FUNCTION_BLOCK XtsMover_TestSuite
VAR
	_TestMoverInterface : I_TcIoXtsXpuMover;
	ThisTestSuite : TestSuite<TestSuiteParameter.MaxTestCount>('C:\ProgramData\Beckhoff\TwinCAT\3.1\Boot\XtsMover_Tests.xml') := (TestSuiteName := 'XtsMover Test Suite');
END_VAR

MoverAcceptsEnableCommand_Test();
MoverAcceptsDisableCommand_Test();
MoverAcceptsGoodGap_Test();
MoverAcceptsModuloBackwardMove_Test();
MoverAcceptsModuloForwardMove_Test();
MoverAcceptsModuloForwardOnlyCommand_Test();
MoverAcceptsNonModuloMoveCommand_Test();
MoverRejectsDisableCommand_Test();
MoverRejectsEnableCommand_Test();
MoverRejectsGapLow_Test();
MoverRejectsHighVeloCommand_Test();
MoverRejectsNegVeloCommand_Test();
MoverRejectsResetWithNoError_Test();
MoverRejectsActivateZeroTrack_Test();
MoverRejectsUnusedHighIndexTrack_Test();
MoverRejectsActivateTrackWhileMoving_Test();
MoverRejectsZeroRefSysWhenMoving_Test();
MoverAcceptsZeroRefSysSet_Test();
MoverRejectsCycleCallWithNoAxisRef_Test();
MoverReportsMovingCorrectly_Test();
MoverReportsMoverOutsidePosWindow_Test();
MoverReportsPositionInWindow_Test();
MoverAcceptsTrackRegistration_Test();
MoverRejectsNullTrackRegister_Test();
MoverRejectsDoubleTrackRegister_Test();
MoverRejectsPosCheckwithNoTrack_Test();
MoverRejectsArriveCommandIfNotLeft_Test();
MoverRejectsArriveCommandIfNoInterface_Test();
MoverRejectsLeaveCommandWithNoInterface_Test();
MoverRejectsLeaveCommandIfMoving_Test();
MoverAcceptsMoverLeaveCommand_Test();
MoverAcceptsArriveCommand_Test();
MoverRejectsAbsMoveToSamePosition();
MoverRejectsModuloMoveToSamePosition();

METHOD MoverAcceptsArriveCommand_Test
VAR_INST
	Expected : BOOL := TRUE;
	Actual	 : BOOL;
END_VAR
VAR
	testMover : stubMover;
END_VAR
IF ThisTestSuite.Test(__POUNAME()).ExecuteTest() THEN
	testMover.MoverXtsIoEnvInterface := _TestMoverInterface;
	Actual := SUCCEEDED(testMover.TriggerMoverArrive());
	ThisTestSuite.Test(__POUNAME()).AssertEqual(Expected, Actual);
END_IF
END_METHOD

METHOD MoverAcceptsDisableCommand_Test
VAR_INST
	Expected : BOOL := TRUE;
	Actual	 : BOOL;
END_VAR
VAR
	testMover : stubMover;
END_VAR
IF ThisTestSuite.Test(__POUNAME()).ExecuteTest() THEN
	testMover.setEnabled();
	Actual := SUCCEEDED( testMover.DisableMover());
	ThisTestSuite.Test(__POUNAME()).AssertEqual(Expected, Actual);
END_IF
END_METHOD

METHOD MoverAcceptsEnableCommand_Test : BOOL
VAR_INST
	Expected : BOOL := TRUE;
	Actual	 : BOOL;
END_VAR
VAR
	testMover : stubMover;
END_VAR
IF ThisTestSuite.Test(__POUNAME()).ExecuteTest() THEN
	testMover.setDisabled();
	Actual := SUCCEEDED( testMover.EnableMover());
	ThisTestSuite.Test(__POUNAME()).AssertEqual(Expected, Actual);
END_IF
END_METHOD

METHOD MoverAcceptsGoodGap_Test : BOOL
VAR_INST
	Expected : mc_lreal := 120.0;
	Actual	 : mc_lreal;
END_VAR
VAR
	testMover : XtsMover;
END_VAR
IF ThisTestSuite.Test(__POUNAME()).ExecuteTest() THEN
	testMover.Gap := 120.0;
	Actual := testMover.Gap;
	ThisTestSuite.Test(__POUNAME()).AssertEqual(Expected, Actual);
END_IF
END_METHOD

METHOD MoverAcceptsModuloBackwardMove_Test
VAR_INST
	Expected : BOOL := TRUE;
	Actual	 : BOOL;
END_VAR
VAR
	testMover : stubMover;
END_VAR
IF ThisTestSuite.Test(__POUNAME()).ExecuteTest() THEN
	testMover.PositiveDirectionOnly := FALSE;
	Actual := testMover.MoveTo(RequiredPosition := - 100.0,
											MoveVelocity := 10.0,
											NonModuloMove := FALSE) = 4;
	ThisTestSuite.Test(__POUNAME()).AssertEqual(Expected, Actual);
END_IF
END_METHOD

METHOD MoverAcceptsModuloForwardMove_Test
VAR_INST
	Expected : BOOL := TRUE;
	Actual	 : BOOL;
END_VAR
VAR
	testMover : stubMover;
END_VAR
IF ThisTestSuite.Test(__POUNAME()).ExecuteTest() THEN
	testMover.PositiveDirectionOnly := FALSE;
	Actual := testMover.MoveTo(RequiredPosition := 100.0,
											MoveVelocity := 10.0,
											NonModuloMove := FALSE) = 3;
	ThisTestSuite.Test(__POUNAME()).AssertEqual(Expected, Actual);
END_IF
END_METHOD

METHOD MoverAcceptsModuloForwardOnlyCommand_Test
VAR_INST
	Expected : BOOL := TRUE;
	Actual	 : BOOL;
END_VAR
VAR
	testMover : stubMover;
END_VAR
IF ThisTestSuite.Test(__POUNAME()).ExecuteTest() THEN
	testMover.PositiveDirectionOnly := TRUE;
	Actual := testMover.MoveTo(RequiredPosition := 100.0,
											MoveVelocity := 10.0,
											NonModuloMove := FALSE) = 2;
	ThisTestSuite.Test(__POUNAME()).AssertEqual(Expected, Actual);
	testMover.PositiveDirectionOnly := FALSE;
END_IF
END_METHOD

METHOD MoverAcceptsMoverLeaveCommand_Test
VAR_INST
	Expected : BOOL := TRUE;
	Actual	 : BOOL;
END_VAR
VAR
	testMover : stubMover;
END_VAR
IF ThisTestSuite.Test(__POUNAME()).ExecuteTest() THEN
	testMover.MoverXtsIoEnvInterface := _TestMoverInterface;
	testMover.setActive();
	testMover.setStationary();
	Actual := SUCCEEDED(testMover.TriggerMoverLeave());
	ThisTestSuite.Test(__POUNAME()).AssertEqual(Expected, Actual);
END_IF
END_METHOD

METHOD MoverAcceptsNonModuloMoveCommand_Test
VAR_INST
	Expected : BOOL := TRUE;
	Actual	 : BOOL;
END_VAR
VAR
	testMover : stubMover;
END_VAR
IF ThisTestSuite.Test(__POUNAME()).ExecuteTest() THEN
	Actual := testMover.MoveTo(RequiredPosition := 100.0,
											MoveVelocity := 10.0,
											NonModuloMove := TRUE) = 1;
	ThisTestSuite.Test(__POUNAME()).AssertEqual(Expected, Actual);
END_IF
END_METHOD

METHOD MoverAcceptsTrackRegistration_Test
VAR_INST
	Expected : BOOL := TRUE;
	Actual	 : BOOL;
END_VAR
VAR
	teststubMover : stubMover;
	stubTrack : XtsTrack('');
END_VAR
IF ThisTestSuite.Test(__POUNAME()).ExecuteTest() THEN
	Actual := SUCCEEDED(teststubMover.RegisterTracks(stubTrack));
	ThisTestSuite.Test(__POUNAME()).AssertEqual(Expected, Actual);
END_IF
END_METHOD

METHOD MoverAcceptsZeroRefSysSet_Test
VAR_INST
	Expected : BOOL := TRUE;
	Actual	 : BOOL;
END_VAR
VAR
	testMover : stubMover;
END_VAR
IF ThisTestSuite.Test(__POUNAME()).ExecuteTest() THEN
	testMover.setEnabled();
	testMover.setStationary();
	Actual := SUCCEEDED( testMover.ActivateZeroReferenceSystem());
	ThisTestSuite.Test(__POUNAME()).AssertEqual(Expected, Actual);
END_IF
END_METHOD

PROPERTY MoverInterface : I_TcIoXtsXpuMover
SET
_TestMoverInterface := MoverInterface;
END_SET
END_PROPERTY

METHOD MoverRejectsAbsMoveToSamePosition
VAR_INST
	Expected : BOOL := TRUE;
	Actual	 : BOOL;
END_VAR
VAR
	testMover : stubMover;
END_VAR
IF ThisTestSuite.Test(__POUNAME()).ExecuteTest() THEN
	testMover.setAAbsPosition(100.0);
	Actual := FAILED( testMover.MoveTo(100.0,-1.0,TRUE));
	ThisTestSuite.Test(__POUNAME()).AssertEqual(Expected, Actual);
END_IF
END_METHOD

METHOD MoverRejectsActivateTrackWhileMoving_Test
VAR_INST
	Expected : BOOL := TRUE;
	Actual	 : BOOL;
END_VAR
VAR
	teststubMover : stubMover;
	stubTrack : XtsTrack('');
END_VAR
IF ThisTestSuite.Test(__POUNAME()).ExecuteTest() THEN
	teststubMover.RegisterTracks(stubTrack);
	teststubMover.setMoving();
	Actual := teststubMover.ActivateTrack(Track := 1) = -3;
	ThisTestSuite.Test(__POUNAME()).AssertEqual(Expected, Actual);
END_IF
END_METHOD

METHOD MoverRejectsActivateZeroTrack_Test : BOOL
VAR_INST
	Expected : BOOL := TRUE;
	Actual	 : BOOL;
END_VAR
VAR
	testMover : XtsMover;
END_VAR
IF ThisTestSuite.Test(__POUNAME()).ExecuteTest() THEN
	Actual := testMover.ActivateTrack(Track := 0) = -1;
	ThisTestSuite.Test(__POUNAME()).AssertEqual(Expected, Actual);
END_IF
END_METHOD

METHOD MoverRejectsArriveCommandIfNoInterface_Test
VAR_INST
	Expected : BOOL := TRUE;
	Actual	 : BOOL;
END_VAR
VAR
	testMover : stubMover;
END_VAR
IF ThisTestSuite.Test(__POUNAME()).ExecuteTest() THEN
	Actual := testMover.TriggerMoverArrive() = -1;
	ThisTestSuite.Test(__POUNAME()).AssertEqual(Expected, Actual);
END_IF
END_METHOD

METHOD MoverRejectsArriveCommandIfNotLeft_Test
VAR_INST
	Expected : BOOL := TRUE;
	Actual	 : BOOL;
END_VAR
VAR
	testMover : stubMover;
END_VAR
IF ThisTestSuite.Test(__POUNAME()).ExecuteTest() THEN
	testMover.setActive();
	testMover.MoverXtsIoEnvInterface := _TestMoverInterface;
	Actual := testMover.TriggerMoverArrive() = -2;
	ThisTestSuite.Test(__POUNAME()).AssertEqual(Expected, Actual);
END_IF
END_METHOD

METHOD MoverRejectsCycleCallWithNoAxisRef_Test : BOOL
VAR_INST
	Expected : BOOL := TRUE;
	Actual	 : BOOL;
END_VAR
VAR
	testMover : XtsMover;
END_VAR
IF ThisTestSuite.Test(__POUNAME()).ExecuteTest() THEN
	Actual := FAILED( testMover.Cycle());
	ThisTestSuite.Test(__POUNAME()).AssertEqual(Expected, Actual);
END_IF
END_METHOD

METHOD MoverRejectsDisableCommand_Test : BOOL
VAR_INST
	Expected : BOOL := TRUE;
	Actual	 : BOOL;
END_VAR
VAR
	testMover : stubMover;
END_VAR
IF ThisTestSuite.Test(__POUNAME()).ExecuteTest() THEN
	testMover.setDisabled();
	Actual := FAILED( testMover.DisableMover());
	ThisTestSuite.Test(__POUNAME()).AssertEqual(Expected, Actual);
END_IF
END_METHOD

METHOD MoverRejectsDoubleTrackRegister_Test
VAR_INST
	Expected : BOOL := TRUE;
	Actual	 : BOOL;
END_VAR
VAR
	teststubMover : stubMover;
	stubTrack : XtsTrack('');
END_VAR
IF ThisTestSuite.Test(__POUNAME()).ExecuteTest() THEN
	teststubMover.RegisterTracks(stubTrack);
	Actual := teststubMover.RegisterTracks(stubTrack) = -2;
	ThisTestSuite.Test(__POUNAME()).AssertEqual(Expected, Actual);
END_IF
END_METHOD

METHOD MoverRejectsEnableCommand_Test
VAR_INST
	Expected : BOOL := TRUE;
	Actual	 : BOOL;
END_VAR
VAR
	testMover : stubMover;
END_VAR
IF ThisTestSuite.Test(__POUNAME()).ExecuteTest() THEN
	testMover.setEnabled();
	Actual := FAILED( testMover.EnableMover());
	ThisTestSuite.Test(__POUNAME()).AssertEqual(Expected, Actual);
END_IF
END_METHOD

METHOD MoverRejectsGapLow_Test : BOOL
VAR_INST
	Expected : mc_lreal := 100.0;
	Actual	 : mc_lreal;
END_VAR
VAR
	testMover : XtsMover;
END_VAR
IF ThisTestSuite.Test(__POUNAME()).ExecuteTest() THEN
	testMover.Gap := 25.0;
	Actual := testMover.Gap;
	ThisTestSuite.Test(__POUNAME()).AssertEqual(Expected, Actual);
END_IF
END_METHOD

METHOD MoverRejectsHighVeloCommand_Test : BOOL
VAR_INST
	Expected : BOOL := TRUE;
	Actual	 : BOOL;
END_VAR
VAR
	testMover : XtsMover;
END_VAR
IF ThisTestSuite.Test(__POUNAME()).ExecuteTest() THEN
	Actual := FAILED( testMover.MoveTo(100.0,5000.0,true));
	ThisTestSuite.Test(__POUNAME()).AssertEqual(Expected, Actual);
END_IF
END_METHOD

METHOD MoverRejectsLeaveCommandIfMoving_Test
VAR_INST
	Expected : BOOL := TRUE;
	Actual	 : BOOL;
END_VAR
VAR
	testMover : stubMover;
END_VAR
IF ThisTestSuite.Test(__POUNAME()).ExecuteTest() THEN
	testMover.setMoving();
	testMover.setActive();
	testMover.MoverXtsIoEnvInterface := _TestMoverInterface;
	Actual := testMover.TriggerMoverLeave() = -3;
	ThisTestSuite.Test(__POUNAME()).AssertEqual(Expected, Actual);
END_IF
END_METHOD

METHOD MoverRejectsLeaveCommandWithNoInterface_Test
VAR_INST
	Expected : BOOL := TRUE;
	Actual	 : BOOL;
END_VAR
VAR
	testMover : stubMover;
END_VAR
IF ThisTestSuite.Test(__POUNAME()).ExecuteTest() THEN
	Actual := testMover.TriggerMoverLeave() = -1;
	ThisTestSuite.Test(__POUNAME()).AssertEqual(Expected, Actual);
END_IF
END_METHOD

METHOD MoverRejectsModuloMoveToSamePosition
VAR_INST
	Expected : BOOL := TRUE;
	Actual	 : BOOL;
END_VAR
VAR
	testMover : stubMover;
END_VAR
IF ThisTestSuite.Test(__POUNAME()).ExecuteTest() THEN
	testMover.setAPosition(100.0);
	Actual := FAILED( testMover.MoveTo(100.0,-1.0,FALSE));
	ThisTestSuite.Test(__POUNAME()).AssertEqual(Expected, Actual);
END_IF
END_METHOD

METHOD MoverRejectsNegVeloCommand_Test : BOOL
VAR_INST
	Expected : BOOL := TRUE;
	Actual	 : BOOL;
END_VAR
VAR
	testMover : XtsMover;
END_VAR
IF ThisTestSuite.Test(__POUNAME()).ExecuteTest() THEN
	Actual := FAILED( testMover.MoveTo(100.0,-1.0,TRUE));
	ThisTestSuite.Test(__POUNAME()).AssertEqual(Expected, Actual);
END_IF
END_METHOD

METHOD MoverRejectsNullTrackRegister_Test
VAR_INST
	Expected : BOOL := TRUE;
	Actual	 : BOOL;
END_VAR
VAR
	teststubMover : stubMover;
	stubTrack : I_XtsTrack;
END_VAR
IF ThisTestSuite.Test(__POUNAME()).ExecuteTest() THEN
	Actual := teststubMover.RegisterTracks(stubTrack) = -1;
	ThisTestSuite.Test(__POUNAME()).AssertEqual(Expected, Actual);
END_IF
END_METHOD

METHOD MoverRejectsPosCheckwithNoTrack_Test
VAR_INST
	Expected : BOOL := TRUE;
	Actual	 : BOOL;
END_VAR
VAR
	testMover : stubMover;
END_VAR
IF ThisTestSuite.Test(__POUNAME()).ExecuteTest() THEN
	Actual := NOT testMover.isMoverAtPosition(0.0);
	ThisTestSuite.Test(__POUNAME()).AssertEqual(Expected, Actual);
END_IF
END_METHOD

METHOD MoverRejectsResetWithNoError_Test : BOOL
VAR_INST
	Expected : BOOL := TRUE;
	Actual	 : BOOL;
END_VAR
VAR
	testMover : XtsMover;
END_VAR
IF ThisTestSuite.Test(__POUNAME()).ExecuteTest() THEN
	Actual := FAILED( testMover.Reset());
	ThisTestSuite.Test(__POUNAME()).AssertEqual(Expected, Actual);
END_IF
END_METHOD

METHOD MoverRejectsUnusedHighIndexTrack_Test
VAR_INST
	Expected : BOOL := TRUE;
	Actual	 : BOOL;
END_VAR
VAR
	testMover : stubMover;
END_VAR
IF ThisTestSuite.Test(__POUNAME()).ExecuteTest() THEN
	testMover.setStationary();
	Actual := testMover.ActivateTrack(Track := 5) = -4;
	ThisTestSuite.Test(__POUNAME()).AssertEqual(Expected, Actual);
END_IF
END_METHOD

METHOD MoverRejectsZeroRefSysWhenMoving_Test
VAR_INST
	Expected : BOOL := TRUE;
	Actual	 : BOOL;
END_VAR
VAR
	testMover : stubMover;
END_VAR
IF ThisTestSuite.Test(__POUNAME()).ExecuteTest() THEN
	testMover.setEnabled();
	testMover.setMoving();
	Actual := testMover.ActivateZeroReferenceSystem() = -2;
	ThisTestSuite.Test(__POUNAME()).AssertEqual(Expected, Actual);
END_IF
END_METHOD

METHOD MoverReportsMoverOutsidePosWindow_Test
VAR_INST
	Expected : BOOL := TRUE;
	Actual	 : BOOL;
END_VAR
VAR
	testMover : stubMover;
END_VAR
IF ThisTestSuite.Test(__POUNAME()).ExecuteTest() THEN
	testMover.setAPosition(301.2);
	Actual := NOT testMover.isMoverAtPosition(300.0);
	ThisTestSuite.Test(__POUNAME()).AssertEqual(Expected, Actual);
END_IF
END_METHOD

METHOD MoverReportsMovingCorrectly_Test
VAR_INST
	Expected : BOOL := TRUE;
	Actual	 : BOOL;
END_VAR
VAR
	testMover : stubMover;
END_VAR
IF ThisTestSuite.Test(__POUNAME()).ExecuteTest() THEN
	testMover.setMoving();
	Actual := NOT testMover.IsStationary;
	testMover.setStationary();
	Actual := Actual AND testMover.IsStationary;
	ThisTestSuite.Test(__POUNAME()).AssertEqual(Expected, Actual);
END_IF
END_METHOD

METHOD MoverReportsPositionInWindow_Test
VAR_INST
	Expected : BOOL := TRUE;
	Actual	 : BOOL;
END_VAR
VAR
	testMover : stubMover;
END_VAR
IF ThisTestSuite.Test(__POUNAME()).ExecuteTest() THEN
	testMover.setAPosition(301.2);
	Actual := testMover.isMoverAtPosition(302.0);
	ThisTestSuite.Test(__POUNAME()).AssertEqual(Expected, Actual);
END_IF
END_METHOD

END_FUNCTION_BLOCK

(* stored: Version 1.1.0.1
   POU XtsMover_TestSuite: Id {35b3f83a-ddd6-49c7-a80a-724734d90825}, SpecialFunc None
   Method MoverAcceptsArriveCommand_Test: Id {22e6417c-6fbd-4ac0-9667-5e84052cd4a6}
   Method MoverAcceptsDisableCommand_Test: Id {f74263e1-f8f8-472b-b7d9-77e272f7e657}
   Method MoverAcceptsEnableCommand_Test: Id {716146c2-e85b-4cfe-8ba6-0d5e0d358526}
   Method MoverAcceptsGoodGap_Test: Id {a49e7a7f-b905-403f-b266-dc77e02f27a1}
   Method MoverAcceptsModuloBackwardMove_Test: Id {f01ead45-02a1-4332-9b35-9dc1d8e90aa5}
   Method MoverAcceptsModuloForwardMove_Test: Id {07afab8a-841c-4fbe-b344-5bbfa5b521c6}
   Method MoverAcceptsModuloForwardOnlyCommand_Test: Id {a64dceeb-4c24-4d38-9111-5e79894157e6}
   Method MoverAcceptsMoverLeaveCommand_Test: Id {63a4cba1-4cae-4219-85d1-5681444a678f}
   Method MoverAcceptsNonModuloMoveCommand_Test: Id {2b00f225-8b8d-421c-b2e9-7d3989986ec2}
   Method MoverAcceptsTrackRegistration_Test: Id {25290b46-6231-42fb-a203-79bee776a0f7}
   Method MoverAcceptsZeroRefSysSet_Test: Id {df519fe2-b659-439f-acdf-e643f50ea61d}
   Property MoverInterface: Id {f0947ece-3c35-4f88-ac1c-7aec4cecfcaa}
   Set Set: Id {42d5a4ab-8220-4929-b77b-834b5cb51aa6}
   Method MoverRejectsAbsMoveToSamePosition: Id {20395d0d-bef3-4c68-ae81-09a57f71f72f}
   Method MoverRejectsActivateTrackWhileMoving_Test: Id {68602ec7-eeb2-48cd-a3a7-de01a20ff851}
   Method MoverRejectsActivateZeroTrack_Test: Id {63f382c0-31c1-4b25-adcd-c20a2309c7b9}
   Method MoverRejectsArriveCommandIfNoInterface_Test: Id {f97f0d65-3de3-442e-93b9-a0e1236e2cf9}
   Method MoverRejectsArriveCommandIfNotLeft_Test: Id {0e69579f-6dca-4b96-be0e-fb9b4ad240f0}
   Method MoverRejectsCycleCallWithNoAxisRef_Test: Id {fb3f91ca-683c-4eda-a124-b2b3567eaec3}
   Method MoverRejectsDisableCommand_Test: Id {61adacd1-bbb3-4810-9e81-807401845494}
   Method MoverRejectsDoubleTrackRegister_Test: Id {b3316b94-62df-4481-b90b-e4fdb0a8771a}
   Method MoverRejectsEnableCommand_Test: Id {27df6825-6795-4e10-9d4e-f3f97002c790}
   Method MoverRejectsGapLow_Test: Id {6530a17d-1991-47b3-b4cb-06ac96089734}
   Method MoverRejectsHighVeloCommand_Test: Id {5ee085d8-22d2-44c9-b967-7741b9170bcb}
   Method MoverRejectsLeaveCommandIfMoving_Test: Id {8be2157e-7677-4ad4-bee0-dd1b09dcf28b}
   Method MoverRejectsLeaveCommandWithNoInterface_Test: Id {c60f29b7-4527-4eb3-87bf-691b0f2f48d3}
   Method MoverRejectsModuloMoveToSamePosition: Id {8153c6df-89da-4493-854f-55394e57a52b}
   Method MoverRejectsNegVeloCommand_Test: Id {64cadcb0-5bf1-4cfd-9d6d-2fa99dffcb0d}
   Method MoverRejectsNullTrackRegister_Test: Id {11ba333d-6ca9-4e64-ab8f-04293121d125}
   Method MoverRejectsPosCheckwithNoTrack_Test: Id {8942dc59-e1b2-4a12-8224-cfcb7ed3188c}
   Method MoverRejectsResetWithNoError_Test: Id {f5425bf8-2274-4dca-931b-4651d9a2101b}
   Method MoverRejectsUnusedHighIndexTrack_Test: Id {aa50061a-5df7-4dfa-887e-ad5a41146b98}
   Method MoverRejectsZeroRefSysWhenMoving_Test: Id {bb153479-b73c-47fe-b92e-239b0e5bd0d4}
   Method MoverReportsMoverOutsidePosWindow_Test: Id {43848fba-d9e9-410c-98a3-0bba057248aa}
   Method MoverReportsMovingCorrectly_Test: Id {2f7e6e28-944b-4700-8c41-7d154cade07a}
   Method MoverReportsPositionInWindow_Test: Id {53afb953-412d-4aa5-b491-ac154905df0d} *)
